
// ===== library types =====

TYPE "QElement"
   STRUCT
      "name" : String[20];
      "type" : Int;
      number : DWord;
      "string" : String[20];
   END_STRUCT;
END_TYPE

TYPE "QElement"
   STRUCT
      "name" : String[20];
      "type" : Int;
      number : DWord;
      "string" : String[20];
   END_STRUCT;
END_TYPE